FUNCTION_BLOCK FB_CB_GridMVCB EXTENDS FB_CB_Base
//////////////////
//  Motorized Circuit Breaker with telecommAND   Requires Open and Close impulsions.
//////////////////

VAR_INPUT PERSISTENT
	// Parameters of the Object (instance/model specific) 
	
END_VAR

VAR_INPUT
	// I/O Inputs              	
		
END_VAR

VAR
	//M_OPENCLOSE VARIABLES//

	
	//M_ALARMMANAGEMENT VARIABLES//
		
	//M_STATEMANAGER VARIABLES//
MesDataExd			: CB_Standard ; 
	// M_EXECUTE VARIABLES //
		
	// EMULATOR //

		
END_VAR

METHOD M_Execute
VAR_INPUT
END_VAR



SUPER^.M_Execute();

// updat.MesDataExd.MesData.to be used in other functions 
MesDataExd.MesData.MesClosed := RS_Emulate.Q1 ;
END_METHOD

END_FUNCTION_BLOCK

(* stored: Version 1.1.0.1, ProductVersion 3.1.4024.6
   POU FB_CB_GridMVCB: Id {2f1df842-dae7-45ec-b2ee-93ec048e558c}, SpecialFunc None
   Method M_Execute: Id {90b54535-d791-4563-8e05-f10f62510456} *)
